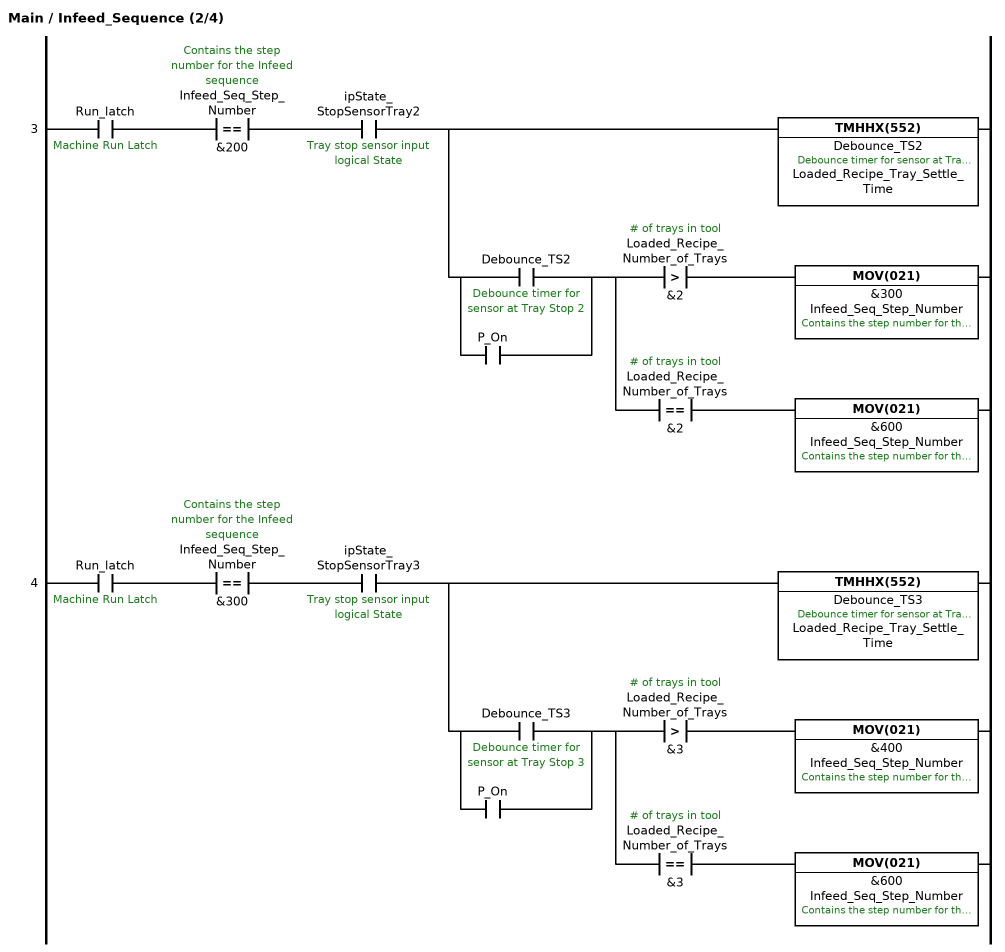
; [picture p24: Main / Infeed_Sequence, rungs 3-4]
; rung 3
LD Run_latch  ; Machine Run Latch
AND=(300) Infeed_Seq_Step_Number &200  ; Contains the step number for the Infeed sequence
AND ipState_StopSensorTray2  ; Tray stop sensor input logical State
TMHHX(552) Debounce_TS2 Loaded_Recipe_Tray_Settle_Time  ; Debounce timer for sensor at Tray Stop 2
LD Debounce_TS2  ; Debounce timer for sensor at Tray Stop 2
OR P_On  // Sensor on and off filters added elsewhere.  Bypassed on 9/25/14 per Gary Liles.
ANDLD
OUT TR0
AND>(320) Loaded_Recipe_Number_of_Trays &2  ; # of trays in tool
MOV(021) &300 Infeed_Seq_Step_Number  ; Contains the step number for the Infeed sequence
LD TR0
AND=(300) Loaded_Recipe_Number_of_Trays &2  ; # of trays in tool
MOV(021) &600 Infeed_Seq_Step_Number  ; Contains the step number for the Infeed sequence
; rung 4
LD Run_latch  ; Machine Run Latch
AND=(300) Infeed_Seq_Step_Number &300  ; Contains the step number for the Infeed sequence
AND ipState_StopSensorTray3  ; Tray stop sensor input logical State
TMHHX(552) Debounce_TS3 Loaded_Recipe_Tray_Settle_Time  ; Debounce timer for sensor at Tray Stop 3
LD Debounce_TS3  ; Debounce timer for sensor at Tray Stop 3
OR P_On  // Sensor on and off filters added elsewhere.  Bypassed on 9/25/14 per Gary Liles.
ANDLD
OUT TR0
AND>(320) Loaded_Recipe_Number_of_Trays &3  ; # of trays in tool
MOV(021) &400 Infeed_Seq_Step_Number  ; Contains the step number for the Infeed sequence
LD TR0
AND=(300) Loaded_Recipe_Number_of_Trays &3  ; # of trays in tool
MOV(021) &600 Infeed_Seq_Step_Number  ; Contains the step number for the Infeed sequence

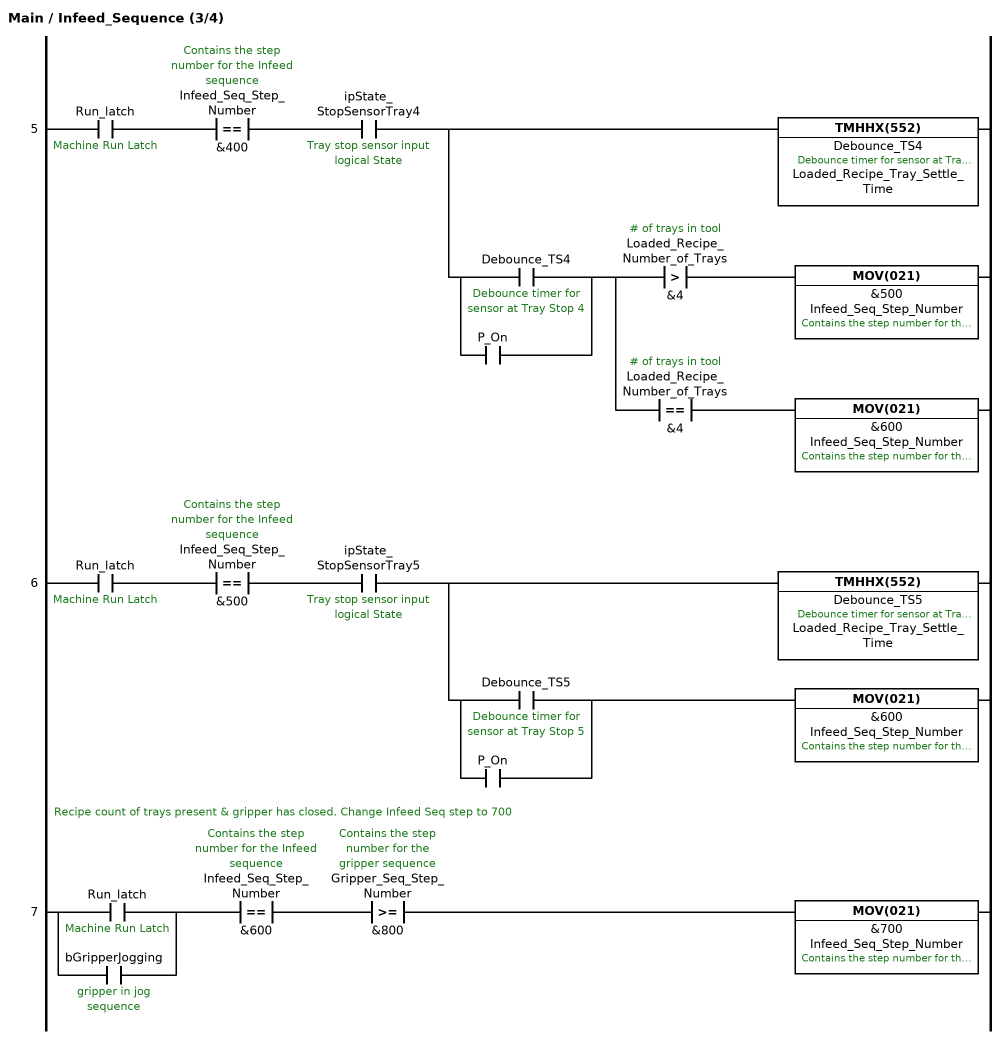
; rung 5
LD Run_latch  ; Machine Run Latch
AND=(300) Infeed_Seq_Step_Number &400  ; Contains the step number for the Infeed sequence
AND ipState_StopSensorTray4  ; Tray stop sensor input logical State
TMHHX(552) Debounce_TS4 Loaded_Recipe_Tray_Settle_Time  ; Debounce timer for sensor at Tray Stop 4
LD Debounce_TS4  ; Debounce timer for sensor at Tray Stop 4
OR P_On  // Sensor on and off filters added elsewhere.  Bypassed on 9/25/14 per Gary Liles.
ANDLD
OUT TR0
AND>(320) Loaded_Recipe_Number_of_Trays &4  ; # of trays in tool
MOV(021) &500 Infeed_Seq_Step_Number  ; Contains the step number for the Infeed sequence
LD TR0
AND=(300) Loaded_Recipe_Number_of_Trays &4  ; # of trays in tool
MOV(021) &600 Infeed_Seq_Step_Number  ; Contains the step number for the Infeed sequence
; rung 6
LD Run_latch  ; Machine Run Latch
AND=(300) Infeed_Seq_Step_Number &500  ; Contains the step number for the Infeed sequence
AND ipState_StopSensorTray5  ; Tray stop sensor input logical State
TMHHX(552) Debounce_TS5 Loaded_Recipe_Tray_Settle_Time  ; Debounce timer for sensor at Tray Stop 5
LD Debounce_TS5  ; Debounce timer for sensor at Tray Stop 5
OR P_On  // Sensor on and off filters added elsewhere.  Bypassed on 9/25/14 per Gary Liles.
ANDLD
MOV(021) &600 Infeed_Seq_Step_Number  ; Contains the step number for the Infeed sequence
; rung 7: Recipe count of trays present & gripper has closed. Change Infeed Seq step to 700
LD Run_latch  ; Machine Run Latch
OR bGripperJogging  ; gripper in jog sequence
AND=(300) Infeed_Seq_Step_Number &600  ; Contains the step number for the Infeed sequence
AND>=(325) Gripper_Seq_Step_Number &800  ; Contains the step number for the gripper sequence
MOV(021) &700 Infeed_Seq_Step_Number  ; Contains the step number for the Infeed sequence

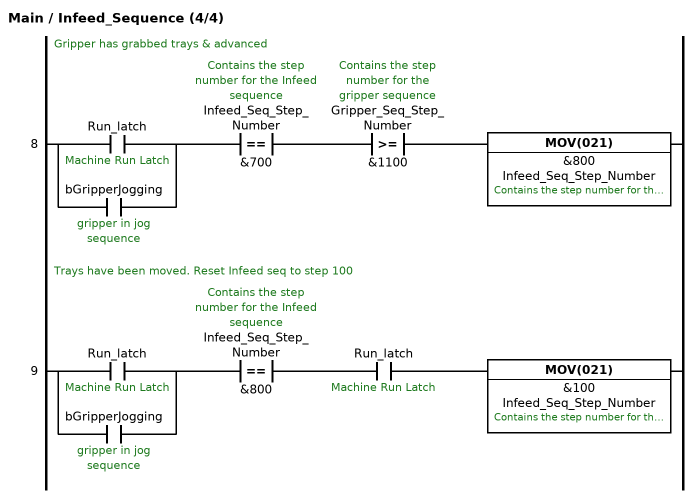
; rung 8: Gripper has grabbed trays & advanced
LD Run_latch  ; Machine Run Latch
OR bGripperJogging  ; gripper in jog sequence
AND=(300) Infeed_Seq_Step_Number &700  ; Contains the step number for the Infeed sequence
AND>=(325) Gripper_Seq_Step_Number &1100  ; Contains the step number for the gripper sequence
MOV(021) &800 Infeed_Seq_Step_Number  ; Contains the step number for the Infeed sequence
; rung 9: Trays have been moved. Reset Infeed seq to step 100
LD Run_latch  ; Machine Run Latch
OR bGripperJogging  ; gripper in jog sequence
AND=(300) Infeed_Seq_Step_Number &800  ; Contains the step number for the Infeed sequence
AND Run_latch  ; Machine Run Latch
MOV(021) &100 Infeed_Seq_Step_Number  ; Contains the step number for the Infeed sequence

### Section Infeed_outputs

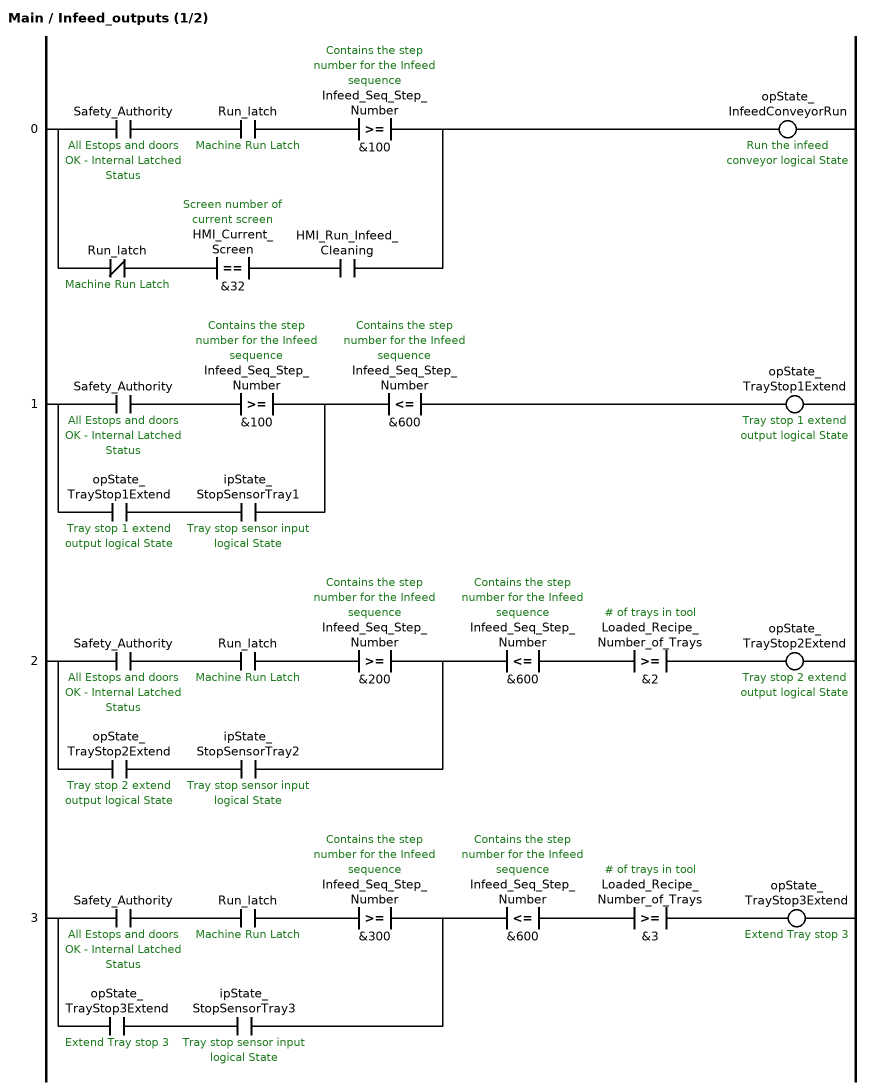
; rung 0
LD Safety_Authority  ; All Estops and doors OK - Internal Latched Status
AND Run_latch  ; Machine Run Latch
AND>=(325) Infeed_Seq_Step_Number &100  ; Contains the step number for the Infeed sequence
LDNOT Run_latch  ; Machine Run Latch
AND=(300) HMI_Current_Screen &32  ; Screen number of current screen
AND HMI_Run_Infeed_Cleaning
ORLD
OUT opState_InfeedConveyorRun  ; Run the infeed conveyor logical State
; rung 1
LD Safety_Authority  ; All Estops and doors OK - Internal Latched Status
AND>=(325) Infeed_Seq_Step_Number &100  ; Contains the step number for the Infeed sequence
LD opState_TrayStop1Extend  ; Tray stop 1 extend output logical State
AND ipState_StopSensorTray1  ; Tray stop sensor input logical State
ORLD
AND<=(315) Infeed_Seq_Step_Number &600  ; Contains the step number for the Infeed sequence
OUT opState_TrayStop1Extend  ; Tray stop 1 extend output logical State
; rung 2
LD Safety_Authority  ; All Estops and doors OK - Internal Latched Status
AND Run_latch  ; Machine Run Latch
AND>=(325) Infeed_Seq_Step_Number &200  ; Contains the step number for the Infeed sequence
LD opState_TrayStop2Extend  ; Tray stop 2 extend output logical State
AND ipState_StopSensorTray2  ; Tray stop sensor input logical State
ORLD
AND<=(315) Infeed_Seq_Step_Number &600  ; Contains the step number for the Infeed sequence
AND>=(325) Loaded_Recipe_Number_of_Trays &2  ; # of trays in tool
OUT opState_TrayStop2Extend  ; Tray stop 2 extend output logical State
; rung 3
LD Safety_Authority  ; All Estops and doors OK - Internal Latched Status
AND Run_latch  ; Machine Run Latch
AND>=(325) Infeed_Seq_Step_Number &300  ; Contains the step number for the Infeed sequence
LD opState_TrayStop3Extend  ; Extend Tray stop 3
AND ipState_StopSensorTray3  ; Tray stop sensor input logical State
ORLD
AND<=(315) Infeed_Seq_Step_Number &600  ; Contains the step number for the Infeed sequence
AND>=(325) Loaded_Recipe_Number_of_Trays &3  ; # of trays in tool
OUT opState_TrayStop3Extend  ; Extend Tray stop 3

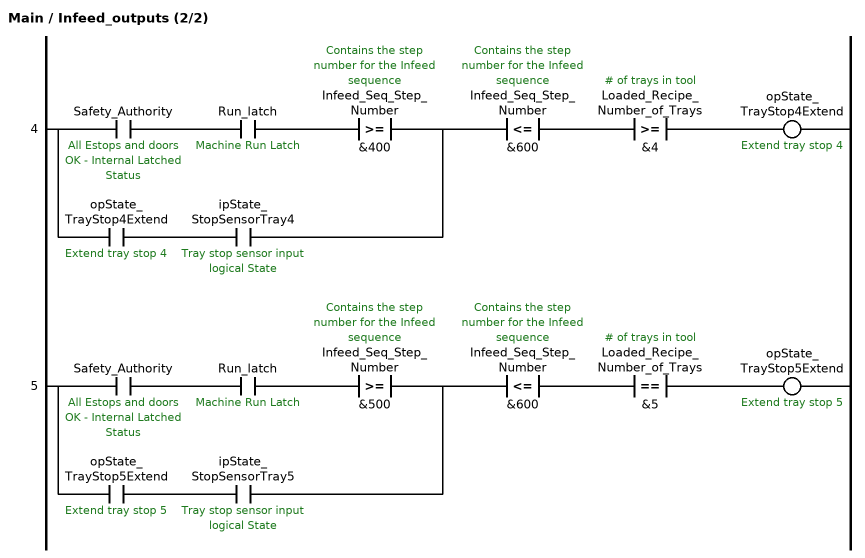
; rung 4
LD Safety_Authority  ; All Estops and doors OK - Internal Latched Status
AND Run_latch  ; Machine Run Latch
AND>=(325) Infeed_Seq_Step_Number &400  ; Contains the step number for the Infeed sequence
LD opState_TrayStop4Extend  ; Extend tray stop 4
AND ipState_StopSensorTray4  ; Tray stop sensor input logical State
ORLD
AND<=(315) Infeed_Seq_Step_Number &600  ; Contains the step number for the Infeed sequence
AND>=(325) Loaded_Recipe_Number_of_Trays &4  ; # of trays in tool
OUT opState_TrayStop4Extend  ; Extend tray stop 4
; rung 5
LD Safety_Authority  ; All Estops and doors OK - Internal Latched Status
AND Run_latch  ; Machine Run Latch
AND>=(325) Infeed_Seq_Step_Number &500  ; Contains the step number for the Infeed sequence
LD opState_TrayStop5Extend  ; Extend tray stop 5
AND ipState_StopSensorTray5  ; Tray stop sensor input logical State
ORLD
AND<=(315) Infeed_Seq_Step_Number &600  ; Contains the step number for the Infeed sequence
AND=(300) Loaded_Recipe_Number_of_Trays &5  ; # of trays in tool
OUT opState_TrayStop5Extend  ; Extend tray stop 5

### Section Grip_Sequence

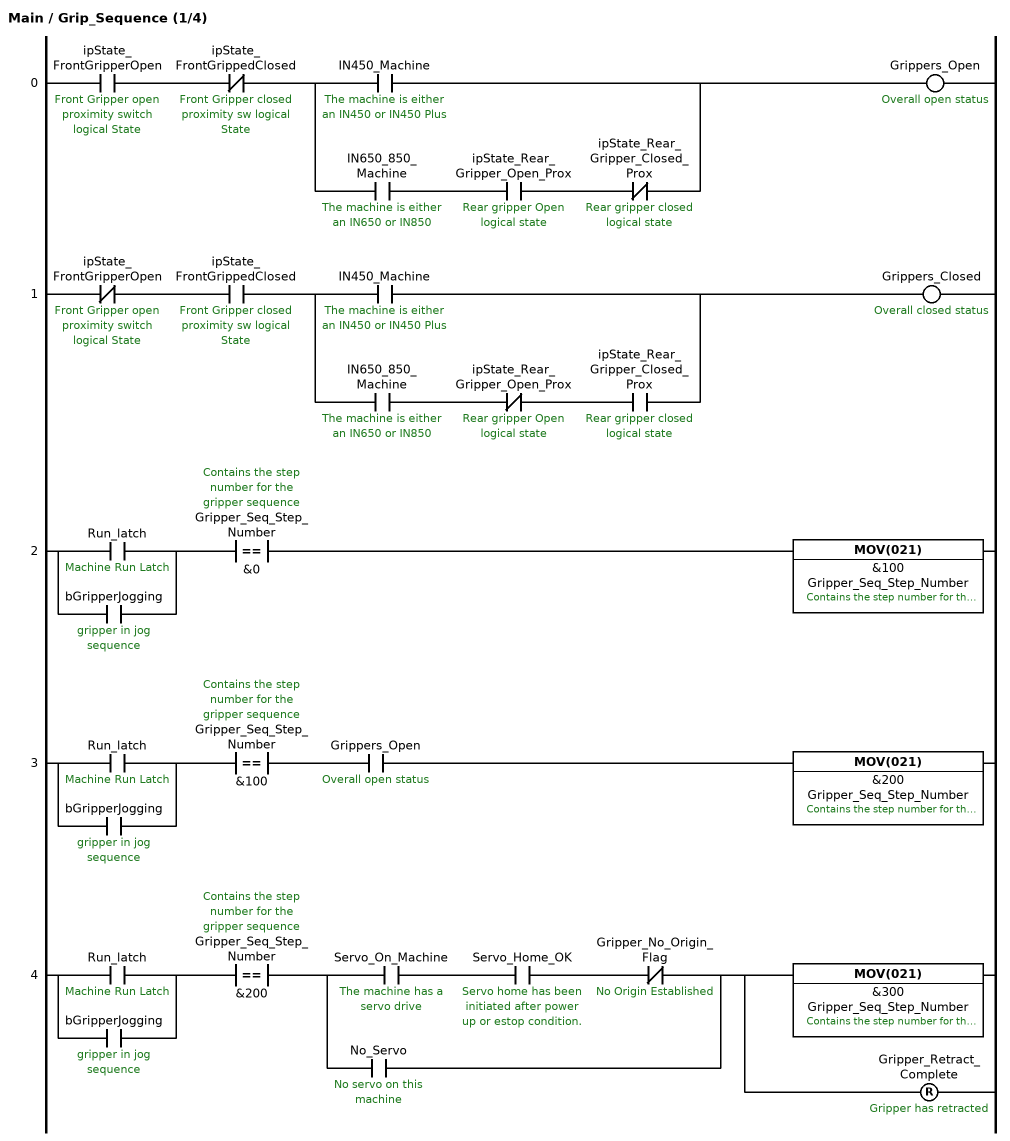
; rung 0
LD ipState_FrontGripperOpen  ; Front Gripper open proximity switch logical State
ANDNOT ipState_FrontGrippedClosed  ; Front Gripper closed proximity sw logical State
LD IN450_Machine  ; The machine is either an IN450 or IN450 Plus
LD IN650_850_Machine  ; The machine is either an IN650 or IN850
AND ipState_Rear_Gripper_Open_Prox  ; Rear gripper Open logical state
ANDNOT ipState_Rear_Gripper_Closed_Prox  ; Rear gripper closed logical state
ORLD
ANDLD
OUT Grippers_Open  ; Overall open status
; rung 1
LDNOT ipState_FrontGripperOpen  ; Front Gripper open proximity switch logical State
AND ipState_FrontGrippedClosed  ; Front Gripper closed proximity sw logical State
LD IN450_Machine  ; The machine is either an IN450 or IN450 Plus
LD IN650_850_Machine  ; The machine is either an IN650 or IN850
ANDNOT ipState_Rear_Gripper_Open_Prox  ; Rear gripper Open logical state
AND ipState_Rear_Gripper_Closed_Prox  ; Rear gripper closed logical state
ORLD
ANDLD
OUT Grippers_Closed  ; Overall closed status
; rung 2
LD Run_latch  ; Machine Run Latch
OR bGripperJogging  ; gripper in jog sequence
AND=(300) Gripper_Seq_Step_Number &0  ; Contains the step number for the gripper sequence
MOV(021) &100 Gripper_Seq_Step_Number  ; Contains the step number for the gripper sequence
; rung 3
LD Run_latch  ; Machine Run Latch
OR bGripperJogging  ; gripper in jog sequence
AND=(300) Gripper_Seq_Step_Number &100  ; Contains the step number for the gripper sequence
AND Grippers_Open  ; Overall open status
MOV(021) &200 Gripper_Seq_Step_Number  ; Contains the step number for the gripper sequence
; rung 4
LD Run_latch  ; Machine Run Latch
OR bGripperJogging  ; gripper in jog sequence
AND=(300) Gripper_Seq_Step_Number &200  ; Contains the step number for the gripper sequence
LD Servo_On_Machine  ; The machine has a servo drive
AND Servo_Home_OK  ; Servo home has been initiated after power up or estop condition.
ANDNOT Gripper_No_Origin_Flag  ; No Origin Established
OR No_Servo  ; No servo on this machine
ANDLD
MOV(021) &300 Gripper_Seq_Step_Number  ; Contains the step number for the gripper sequence
RSET Gripper_Retract_Complete  ; Gripper has retracted

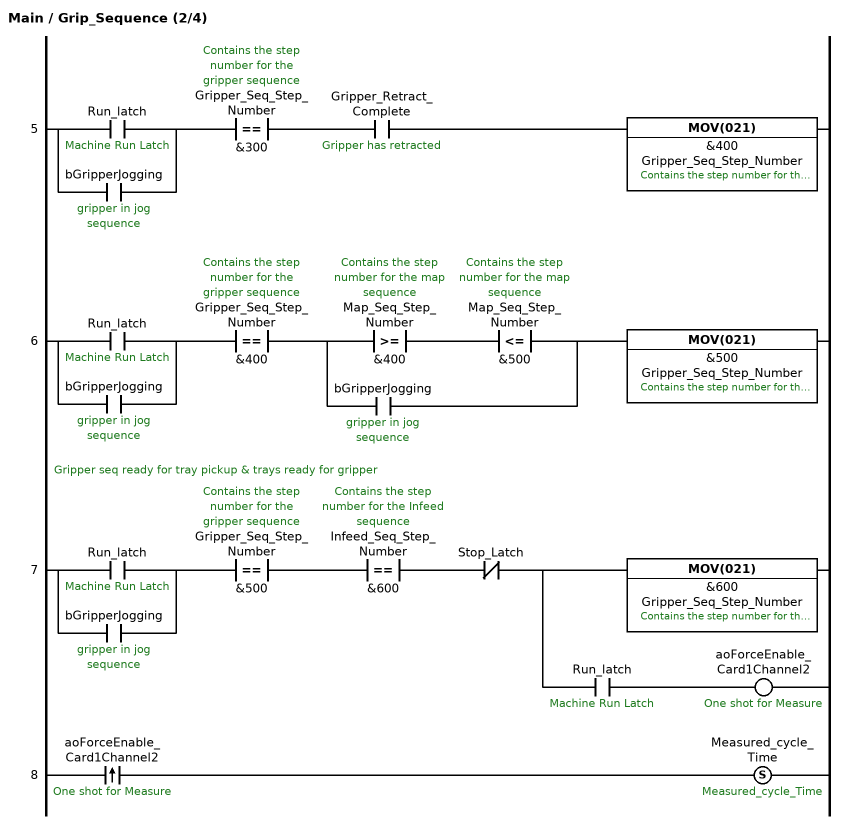
; rung 5
LD Run_latch  ; Machine Run Latch
OR bGripperJogging  ; gripper in jog sequence
AND=(300) Gripper_Seq_Step_Number &300  ; Contains the step number for the gripper sequence
AND Gripper_Retract_Complete  ; Gripper has retracted
MOV(021) &400 Gripper_Seq_Step_Number  ; Contains the step number for the gripper sequence
; rung 6
LD Run_latch  ; Machine Run Latch
OR bGripperJogging  ; gripper in jog sequence
AND=(300) Gripper_Seq_Step_Number &400  ; Contains the step number for the gripper sequence
LD>=(325) Map_Seq_Step_Number &400  ; Contains the step number for the map sequence
AND<=(315) Map_Seq_Step_Number &500  ; Contains the step number for the map sequence
OR bGripperJogging  ; gripper in jog sequence
ANDLD
MOV(021) &500 Gripper_Seq_Step_Number  ; Contains the step number for the gripper sequence
; rung 7: Gripper seq ready for tray pickup & trays ready for gripper
LD Run_latch  ; Machine Run Latch
OR bGripperJogging  ; gripper in jog sequence
AND=(300) Gripper_Seq_Step_Number &500  ; Contains the step number for the gripper sequence
AND=(300) Infeed_Seq_Step_Number &600  ; Contains the step number for the Infeed sequence
ANDNOT Stop_Latch
MOV(021) &600 Gripper_Seq_Step_Number  ; Contains the step number for the gripper sequence
AND Run_latch  ; Machine Run Latch
OUT aoForceEnable_Card1Channel2  ; One shot for Measure
; rung 8
@LD aoForceEnable_Card1Channel2  ; One shot for Measure
SET Measured_cycle_Time  ; Measured_cycle_Time

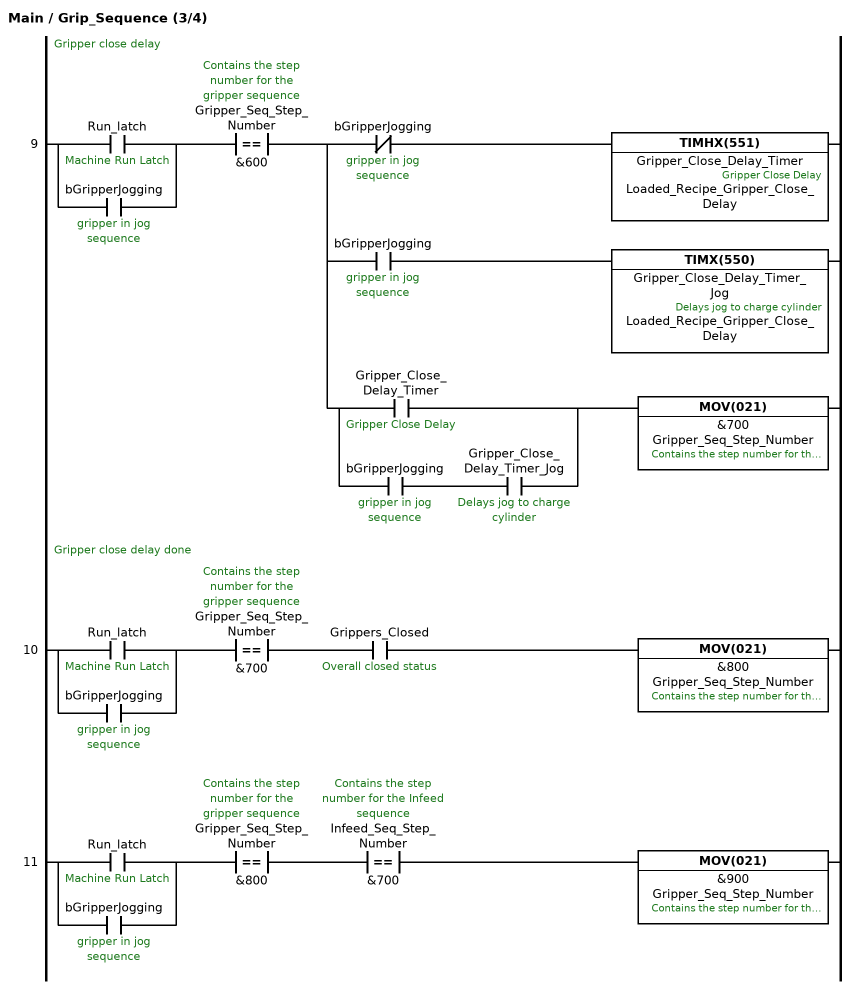
; rung 9: Gripper close delay
LD Run_latch  ; Machine Run Latch
OR bGripperJogging  ; gripper in jog sequence
AND=(300) Gripper_Seq_Step_Number &600  ; Contains the step number for the gripper sequence
OUT TR0
ANDNOT bGripperJogging  ; gripper in jog sequence
TIMHX(551) Gripper_Close_Delay_Timer Loaded_Recipe_Gripper_Close_Delay  ; Gripper Close Delay
LD TR0
AND bGripperJogging  ; gripper in jog sequence
TIMX(550) Gripper_Close_Delay_Timer_Jog Loaded_Recipe_Gripper_Close_Delay  ; Delays jog to charge cylinder
LD TR0
LD Gripper_Close_Delay_Timer  ; Gripper Close Delay
LD bGripperJogging  ; gripper in jog sequence
AND Gripper_Close_Delay_Timer_Jog  ; Delays jog to charge cylinder
ORLD
ANDLD
MOV(021) &700 Gripper_Seq_Step_Number  ; Contains the step number for the gripper sequence
; rung 10: Gripper close delay done
LD Run_latch  ; Machine Run Latch
OR bGripperJogging  ; gripper in jog sequence
AND=(300) Gripper_Seq_Step_Number &700  ; Contains the step number for the gripper sequence
AND Grippers_Closed  ; Overall closed status
MOV(021) &800 Gripper_Seq_Step_Number  ; Contains the step number for the gripper sequence
; rung 11
LD Run_latch  ; Machine Run Latch
OR bGripperJogging  ; gripper in jog sequence
AND=(300) Gripper_Seq_Step_Number &800  ; Contains the step number for the gripper sequence
AND=(300) Infeed_Seq_Step_Number &700  ; Contains the step number for the Infeed sequence
MOV(021) &900 Gripper_Seq_Step_Number  ; Contains the step number for the gripper sequence

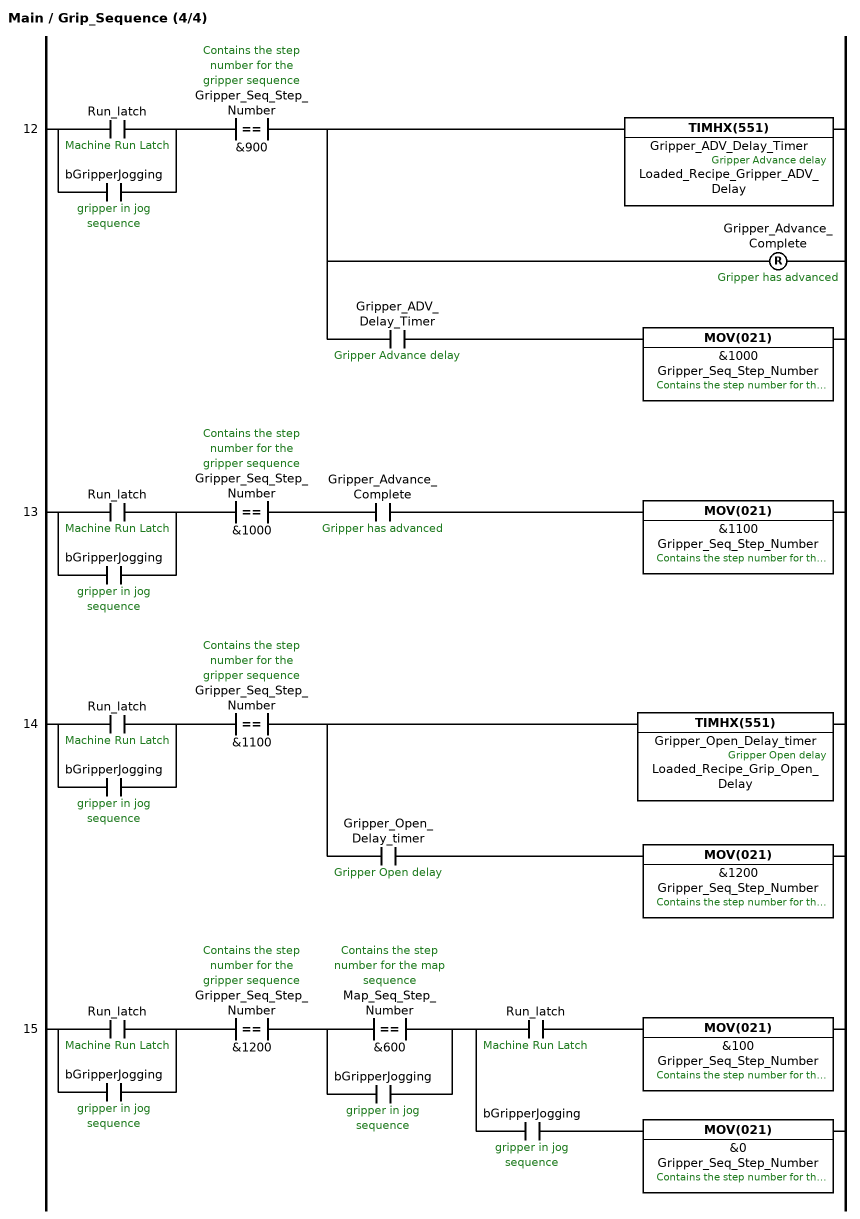
; rung 12
LD Run_latch  ; Machine Run Latch
OR bGripperJogging  ; gripper in jog sequence
AND=(300) Gripper_Seq_Step_Number &900  ; Contains the step number for the gripper sequence
TIMHX(551) Gripper_ADV_Delay_Timer Loaded_Recipe_Gripper_ADV_Delay  ; Gripper Advance delay
RSET Gripper_Advance_Complete  ; Gripper has advanced
AND Gripper_ADV_Delay_Timer  ; Gripper Advance delay
MOV(021) &1000 Gripper_Seq_Step_Number  ; Contains the step number for the gripper sequence
; rung 13
LD Run_latch  ; Machine Run Latch
OR bGripperJogging  ; gripper in jog sequence
AND=(300) Gripper_Seq_Step_Number &1000  ; Contains the step number for the gripper sequence
AND Gripper_Advance_Complete  ; Gripper has advanced
MOV(021) &1100 Gripper_Seq_Step_Number  ; Contains the step number for the gripper sequence
; rung 14
LD Run_latch  ; Machine Run Latch
OR bGripperJogging  ; gripper in jog sequence
AND=(300) Gripper_Seq_Step_Number &1100  ; Contains the step number for the gripper sequence
TIMHX(551) Gripper_Open_Delay_timer Loaded_Recipe_Grip_Open_Delay  ; Gripper Open delay
AND Gripper_Open_Delay_timer  ; Gripper Open delay
MOV(021) &1200 Gripper_Seq_Step_Number  ; Contains the step number for the gripper sequence
; rung 15
LD Run_latch  ; Machine Run Latch
OR bGripperJogging  ; gripper in jog sequence
AND=(300) Gripper_Seq_Step_Number &1200  ; Contains the step number for the gripper sequence
LD=(300) Map_Seq_Step_Number &600  ; Contains the step number for the map sequence
OR bGripperJogging  ; gripper in jog sequence
ANDLD
OUT TR0
AND Run_latch  ; Machine Run Latch
MOV(021) &100 Gripper_Seq_Step_Number  ; Contains the step number for the gripper sequence
LD TR0
AND bGripperJogging  ; gripper in jog sequence
MOV(021) &0 Gripper_Seq_Step_Number  ; Contains the step number for the gripper sequence

### Section Grip_Outputs

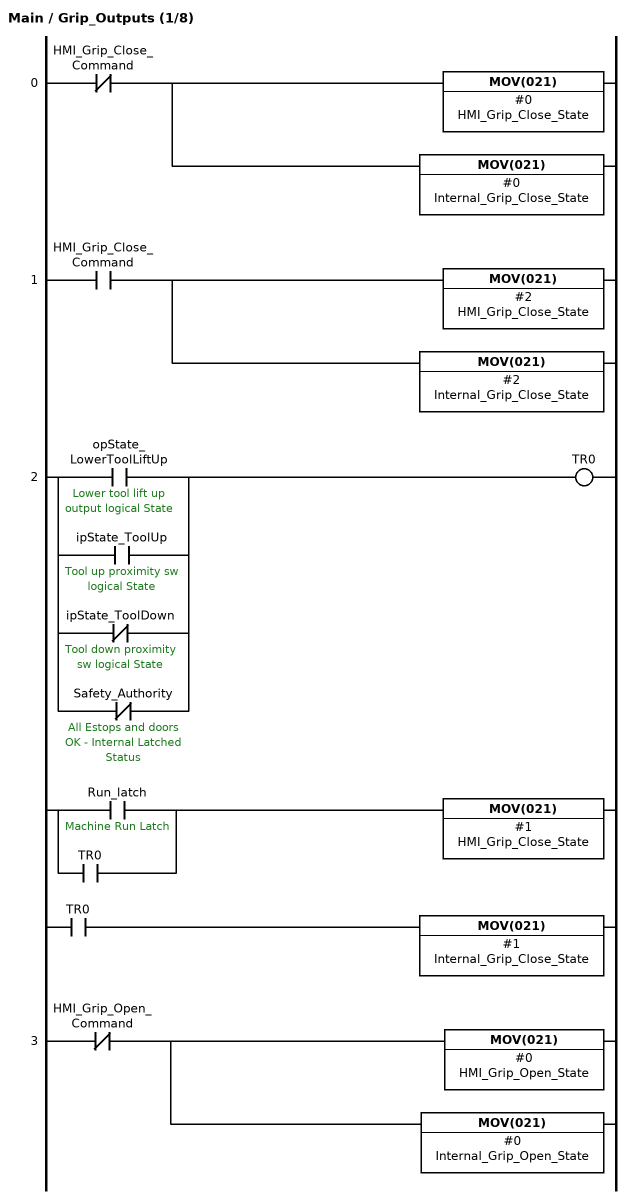
; rung 0
LDNOT HMI_Grip_Close_Command
MOV(021) #0 HMI_Grip_Close_State
MOV(021) #0 Internal_Grip_Close_State
; rung 1
LD HMI_Grip_Close_Command
MOV(021) #2 HMI_Grip_Close_State
MOV(021) #2 Internal_Grip_Close_State
; rung 2
LD Run_latch  ; Machine Run Latch
LD opState_LowerToolLiftUp  ; Lower tool lift up output logical State
OR ipState_ToolUp  ; Tool up proximity sw logical State
ORNOT ipState_ToolDown  ; Tool down proximity sw logical State
ORNOT Safety_Authority  ; All Estops and doors OK - Internal Latched Status
OUT TR0
ORLD
MOV(021) #1 HMI_Grip_Close_State
LD TR0
MOV(021) #1 Internal_Grip_Close_State
; rung 3
LDNOT HMI_Grip_Open_Command
MOV(021) #0 HMI_Grip_Open_State
MOV(021) #0 Internal_Grip_Open_State

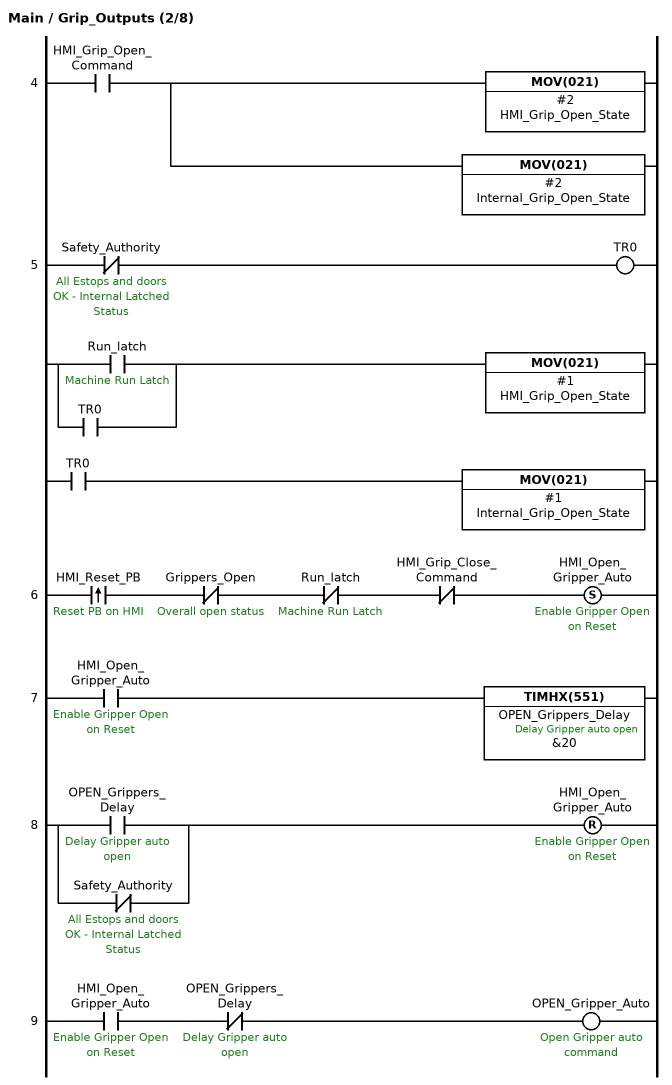
; rung 4
LD HMI_Grip_Open_Command
MOV(021) #2 HMI_Grip_Open_State
MOV(021) #2 Internal_Grip_Open_State
; rung 5
LD Run_latch  ; Machine Run Latch
LDNOT Safety_Authority  ; All Estops and doors OK - Internal Latched Status
OUT TR0
ORLD
MOV(021) #1 HMI_Grip_Open_State
LD TR0
MOV(021) #1 Internal_Grip_Open_State
; rung 6
@LD HMI_Reset_PB  ; Reset PB on HMI
ANDNOT Grippers_Open  ; Overall open status
ANDNOT Run_latch  ; Machine Run Latch
ANDNOT HMI_Grip_Close_Command
SET HMI_Open_Gripper_Auto  ; Enable Gripper Open on Reset
; rung 7
LD HMI_Open_Gripper_Auto  ; Enable Gripper Open on Reset
TIMHX(551) OPEN_Grippers_Delay &20  ; Delay Gripper auto open
; rung 8
LD OPEN_Grippers_Delay  ; Delay Gripper auto open
ORNOT Safety_Authority  ; All Estops and doors OK - Internal Latched Status
RSET HMI_Open_Gripper_Auto  ; Enable Gripper Open on Reset
; rung 9
LD HMI_Open_Gripper_Auto  ; Enable Gripper Open on Reset
ANDNOT OPEN_Grippers_Delay  ; Delay Gripper auto open
OUT OPEN_Gripper_Auto  ; Open Gripper auto command

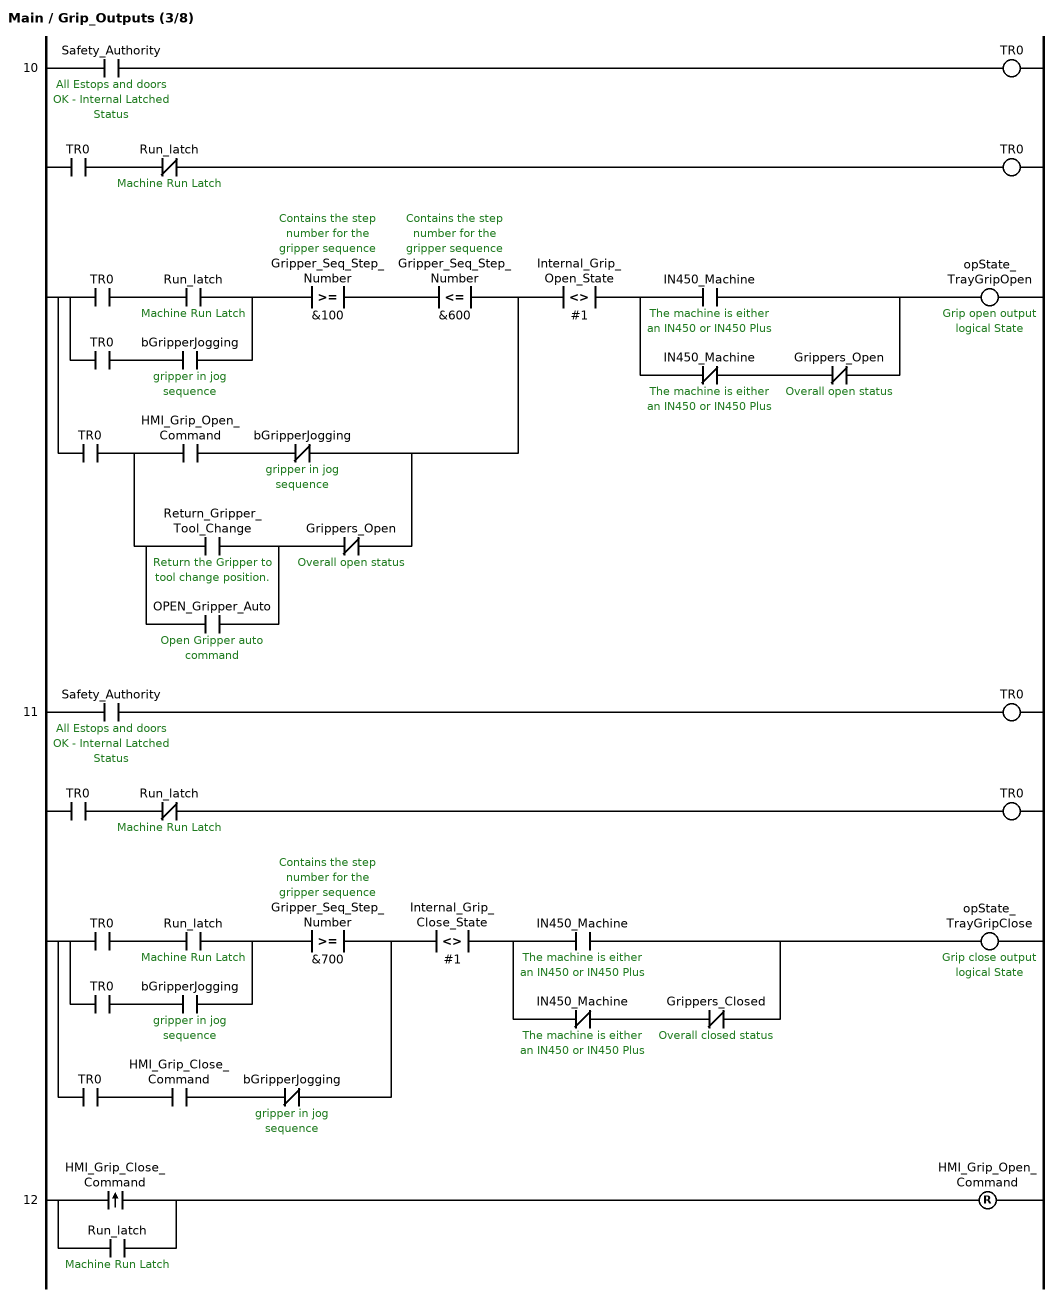
; rung 10
LD Safety_Authority  ; All Estops and doors OK - Internal Latched Status
OUT TR0
AND Run_latch  ; Machine Run Latch
LD TR0
ANDNOT Run_latch  ; Machine Run Latch
OUT TR0
AND bGripperJogging  ; gripper in jog sequence
ORLD
AND>=(325) Gripper_Seq_Step_Number &100  ; Contains the step number for the gripper sequence
AND<=(315) Gripper_Seq_Step_Number &600  ; Contains the step number for the gripper sequence
LD TR0
LD HMI_Grip_Open_Command
ANDNOT bGripperJogging  ; gripper in jog sequence
LD Return_Gripper_Tool_Change  ; Return the Gripper to tool change position.
OR OPEN_Gripper_Auto  ; Open Gripper auto command
ANDNOT Grippers_Open  ; Overall open status
ORLD
ANDLD
ORLD
AND<>(305) Internal_Grip_Open_State #1
LD IN450_Machine  ; The machine is either an IN450 or IN450 Plus
LDNOT IN450_Machine  ; The machine is either an IN450 or IN450 Plus
ANDNOT Grippers_Open  ; Overall open status
ORLD
ANDLD
OUT opState_TrayGripOpen  ; Grip open output logical State
; rung 11
LD Safety_Authority  ; All Estops and doors OK - Internal Latched Status
OUT TR0
AND Run_latch  ; Machine Run Latch
LD TR0
ANDNOT Run_latch  ; Machine Run Latch
OUT TR0
AND bGripperJogging  ; gripper in jog sequence
ORLD
AND>=(325) Gripper_Seq_Step_Number &700  ; Contains the step number for the gripper sequence
LD TR0
AND HMI_Grip_Close_Command
ANDNOT bGripperJogging  ; gripper in jog sequence
ORLD
AND<>(305) Internal_Grip_Close_State #1
LD IN450_Machine  ; The machine is either an IN450 or IN450 Plus
LDNOT IN450_Machine  ; The machine is either an IN450 or IN450 Plus
ANDNOT Grippers_Closed  ; Overall closed status
ORLD
ANDLD
OUT opState_TrayGripClose  ; Grip close output logical State
; rung 12
@LD HMI_Grip_Close_Command
OR Run_latch  ; Machine Run Latch
RSET HMI_Grip_Open_Command

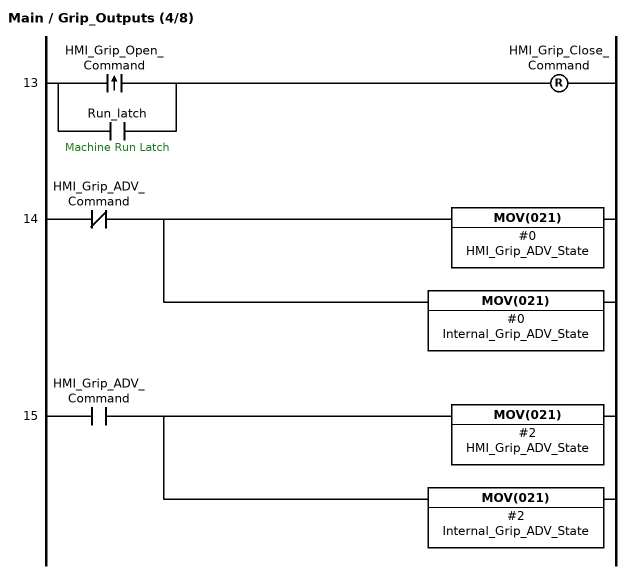
; rung 13
@LD HMI_Grip_Open_Command
OR Run_latch  ; Machine Run Latch
RSET HMI_Grip_Close_Command
; rung 14
LDNOT HMI_Grip_ADV_Command
MOV(021) #0 HMI_Grip_ADV_State
MOV(021) #0 Internal_Grip_ADV_State
; rung 15
LD HMI_Grip_ADV_Command
MOV(021) #2 HMI_Grip_ADV_State
MOV(021) #2 Internal_Grip_ADV_State

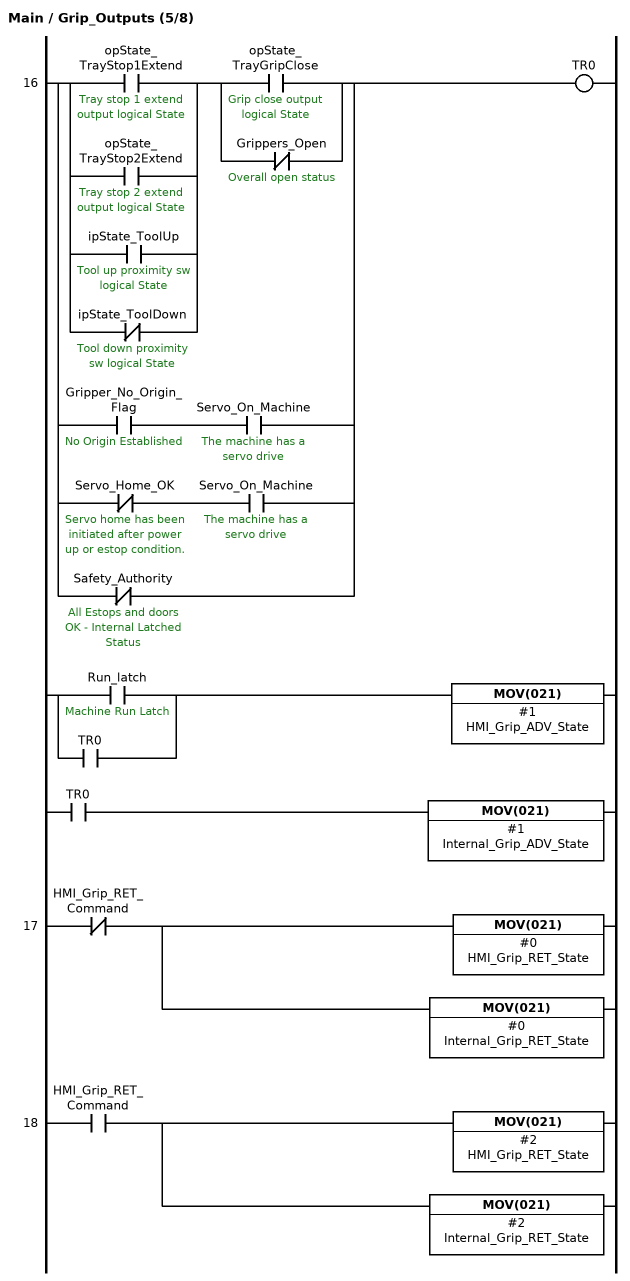
; rung 16
LD Run_latch  ; Machine Run Latch
LD opState_TrayStop1Extend  ; Tray stop 1 extend output logical State
OR opState_TrayStop2Extend  ; Tray stop 2 extend output logical State
OR ipState_ToolUp  ; Tool up proximity sw logical State
ORNOT ipState_ToolDown  ; Tool down proximity sw logical State
LD opState_TrayGripClose  ; Grip close output logical State
ORNOT Grippers_Open  ; Overall open status
ANDLD
LD Gripper_No_Origin_Flag  ; No Origin Established
AND Servo_On_Machine  ; The machine has a servo drive
ORLD
LDNOT Servo_Home_OK  ; Servo home has been initiated after power up or estop condition.
AND Servo_On_Machine  ; The machine has a servo drive
ORLD
ORNOT Safety_Authority  ; All Estops and doors OK - Internal Latched Status
OUT TR0
ORLD
MOV(021) #1 HMI_Grip_ADV_State
LD TR0
MOV(021) #1 Internal_Grip_ADV_State
; rung 17
LDNOT HMI_Grip_RET_Command
MOV(021) #0 HMI_Grip_RET_State
MOV(021) #0 Internal_Grip_RET_State
; rung 18
LD HMI_Grip_RET_Command
MOV(021) #2 HMI_Grip_RET_State
MOV(021) #2 Internal_Grip_RET_State

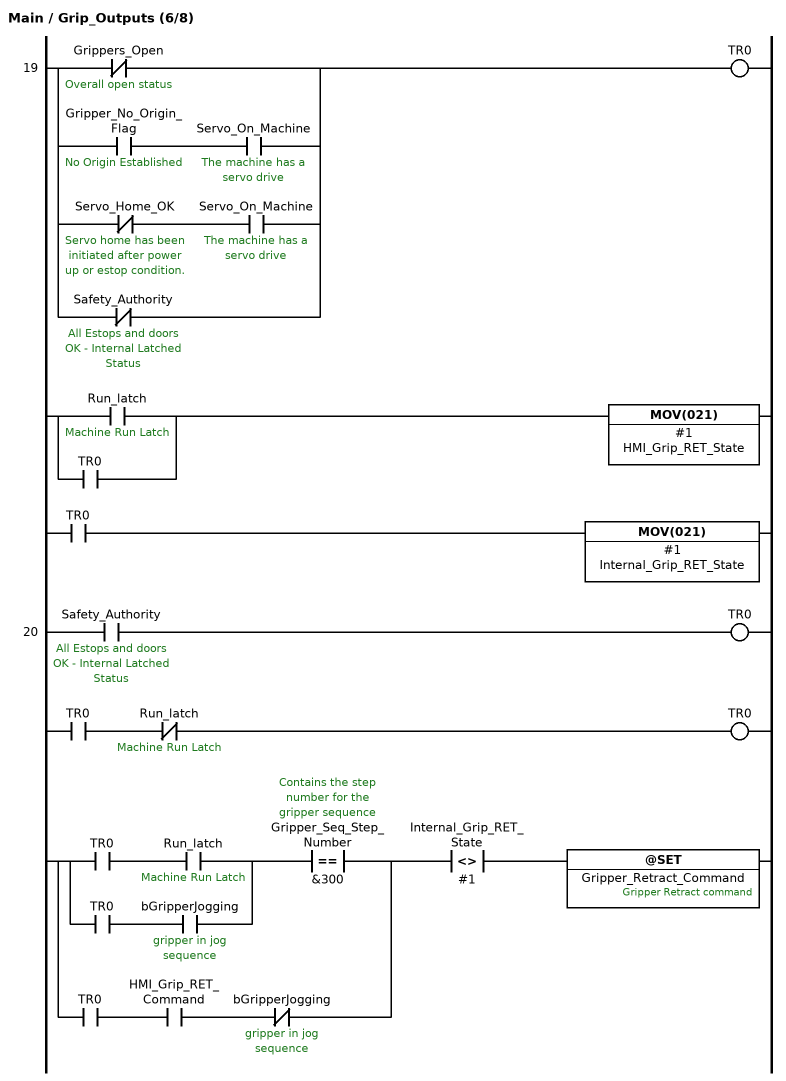
; rung 19
LD Run_latch  ; Machine Run Latch
LDNOT Grippers_Open  ; Overall open status
LD Gripper_No_Origin_Flag  ; No Origin Established
AND Servo_On_Machine  ; The machine has a servo drive
ORLD
LDNOT Servo_Home_OK  ; Servo home has been initiated after power up or estop condition.
AND Servo_On_Machine  ; The machine has a servo drive
ORLD
ORNOT Safety_Authority  ; All Estops and doors OK - Internal Latched Status
OUT TR0
ORLD
MOV(021) #1 HMI_Grip_RET_State
LD TR0
MOV(021) #1 Internal_Grip_RET_State
; rung 20
LD Safety_Authority  ; All Estops and doors OK - Internal Latched Status
OUT TR0
AND Run_latch  ; Machine Run Latch
LD TR0
ANDNOT Run_latch  ; Machine Run Latch
OUT TR0
AND bGripperJogging  ; gripper in jog sequence
ORLD
AND=(300) Gripper_Seq_Step_Number &300  ; Contains the step number for the gripper sequence
LD TR0
AND HMI_Grip_RET_Command
ANDNOT bGripperJogging  ; gripper in jog sequence
ORLD
AND<>(305) Internal_Grip_RET_State #1
@SET Gripper_Retract_Command  ; Gripper Retract command

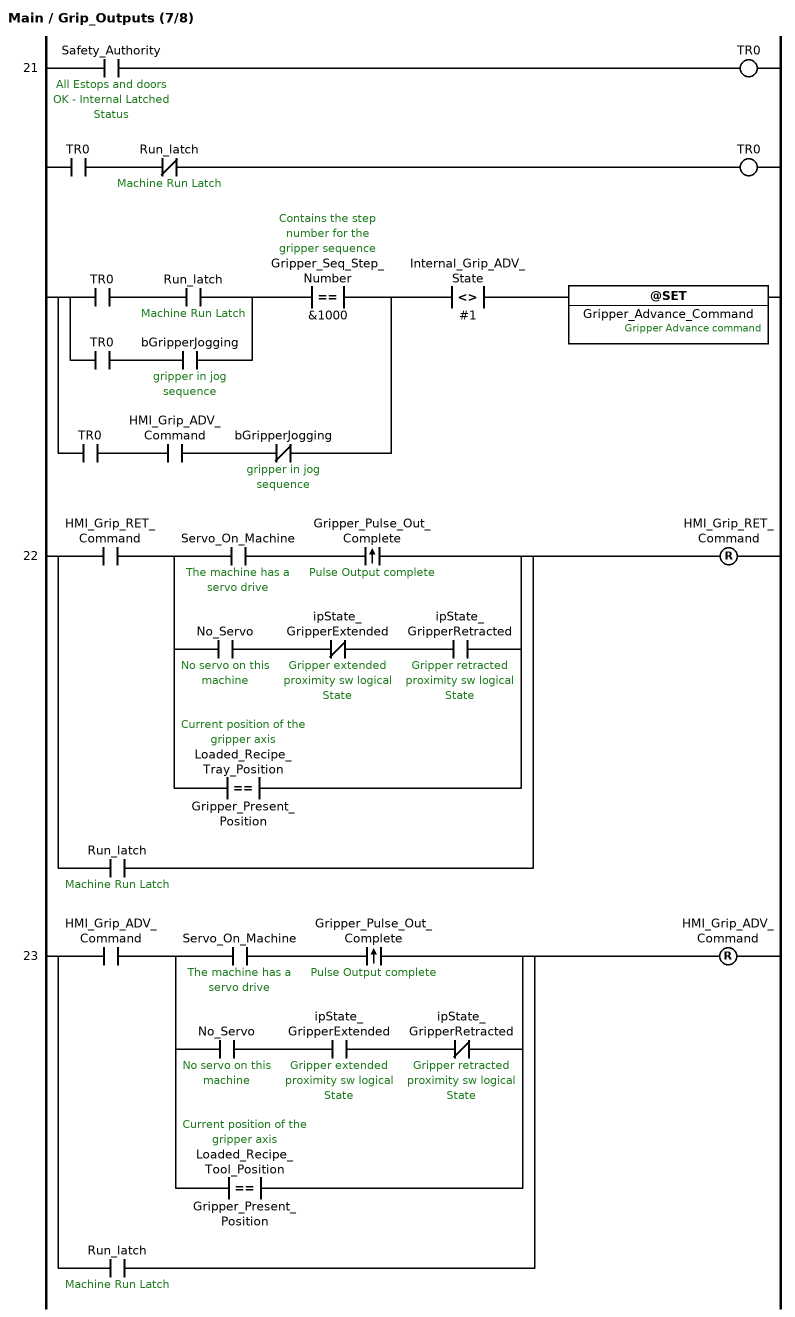
; rung 21
LD Safety_Authority  ; All Estops and doors OK - Internal Latched Status
OUT TR0
AND Run_latch  ; Machine Run Latch
LD TR0
ANDNOT Run_latch  ; Machine Run Latch
OUT TR0
AND bGripperJogging  ; gripper in jog sequence
ORLD
AND=(300) Gripper_Seq_Step_Number &1000  ; Contains the step number for the gripper sequence
LD TR0
AND HMI_Grip_ADV_Command
ANDNOT bGripperJogging  ; gripper in jog sequence
ORLD
AND<>(305) Internal_Grip_ADV_State #1
@SET Gripper_Advance_Command  ; Gripper Advance command
; rung 22
LD HMI_Grip_RET_Command
LD Servo_On_Machine  ; The machine has a servo drive
@AND Gripper_Pulse_Out_Complete  ; Pulse Output complete
LD No_Servo  ; No servo on this machine
ANDNOT ipState_GripperExtended  ; Gripper extended proximity sw logical State
AND ipState_GripperRetracted  ; Gripper retracted proximity sw logical State
ORLD
OR=(300) Loaded_Recipe_Tray_Position Gripper_Present_Position  ; Current position of the gripper axis
ANDLD
OR Run_latch  ; Machine Run Latch
RSET HMI_Grip_RET_Command
; rung 23
LD HMI_Grip_ADV_Command
LD Servo_On_Machine  ; The machine has a servo drive
@AND Gripper_Pulse_Out_Complete  ; Pulse Output complete
LD No_Servo  ; No servo on this machine
AND ipState_GripperExtended  ; Gripper extended proximity sw logical State
ANDNOT ipState_GripperRetracted  ; Gripper retracted proximity sw logical State
ORLD
OR=(300) Loaded_Recipe_Tool_Position Gripper_Present_Position  ; Current position of the gripper axis
ANDLD
OR Run_latch  ; Machine Run Latch
RSET HMI_Grip_ADV_Command

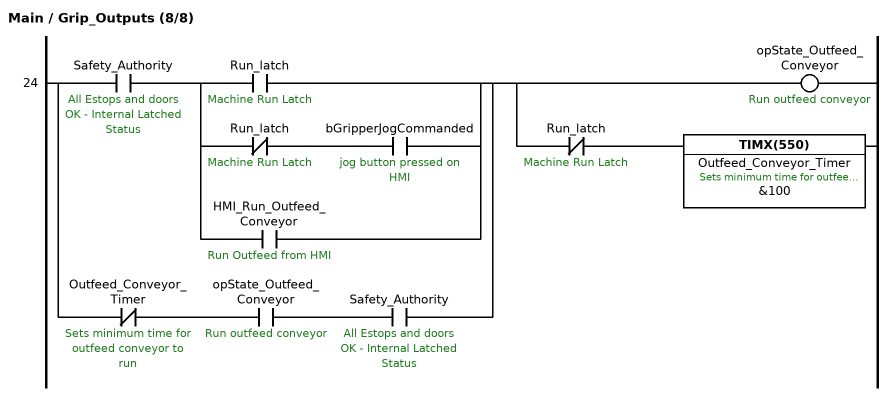
; rung 24
LD Safety_Authority  ; All Estops and doors OK - Internal Latched Status
LD Run_latch  ; Machine Run Latch
LDNOT Run_latch  ; Machine Run Latch
AND bGripperJogCommanded  ; jog button pressed on HMI
ORLD
OR HMI_Run_Outfeed_Conveyor  ; Run Outfeed from HMI
ANDLD
LDNOT Outfeed_Conveyor_Timer  ; Sets minimum time for outfeed conveyor to run
AND opState_Outfeed_Conveyor  ; Run outfeed conveyor
AND Safety_Authority  ; All Estops and doors OK - Internal Latched Status
ORLD
OUT opState_Outfeed_Conveyor  ; Run outfeed conveyor
ANDNOT Run_latch  ; Machine Run Latch
TIMX(550) Outfeed_Conveyor_Timer &100  ; Sets minimum time for outfeed conveyor to run

### Section Infeed_Gate_Sequence

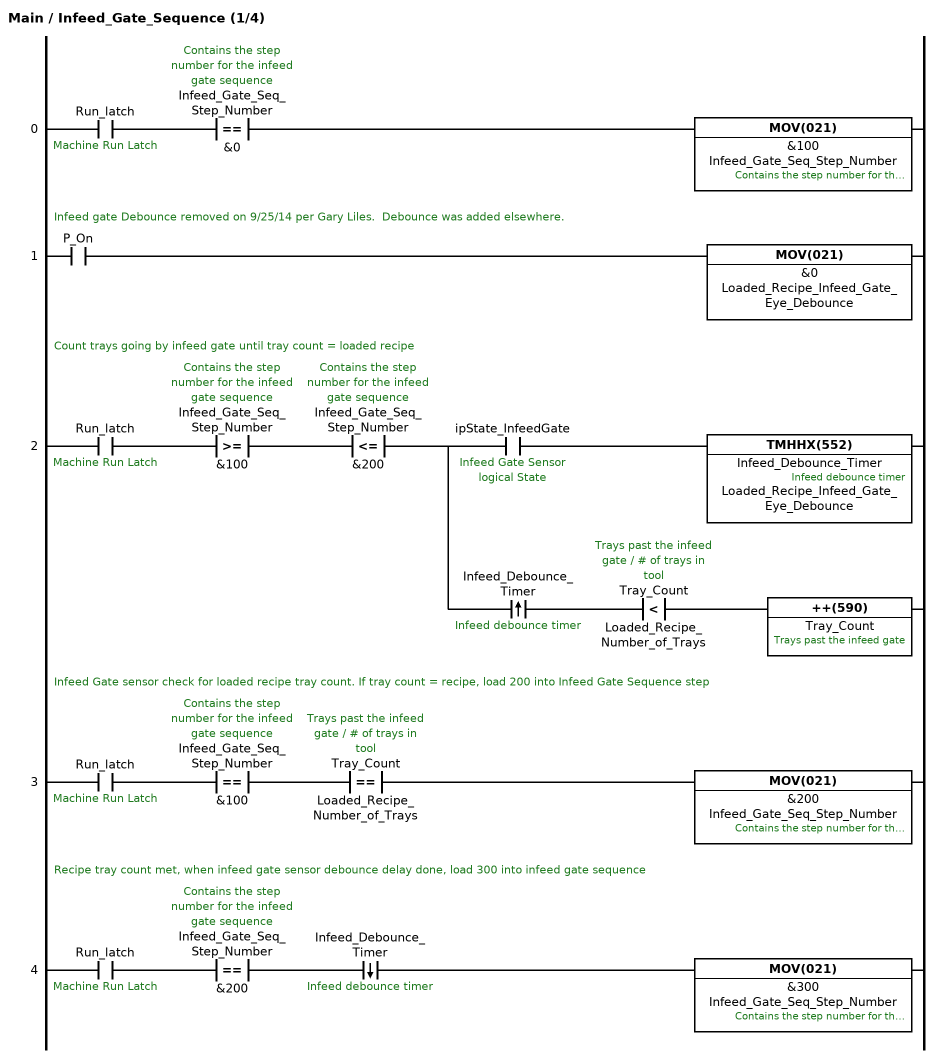
; rung 0
LD Run_latch  ; Machine Run Latch
AND=(300) Infeed_Gate_Seq_Step_Number &0  ; Contains the step number for the infeed gate sequence
MOV(021) &100 Infeed_Gate_Seq_Step_Number  ; Contains the step number for the infeed gate sequence
; rung 1: Infeed gate Debounce removed on 9/25/14 per Gary Liles.  Debounce was added elsewhere.
LD P_On
MOV(021) &0 Loaded_Recipe_Infeed_Gate_Eye_Debounce
; rung 2: Count trays going by infeed gate until tray count = loaded recipe
LD Run_latch  ; Machine Run Latch
AND>=(325) Infeed_Gate_Seq_Step_Number &100  ; Contains the step number for the infeed gate sequence
AND<=(315) Infeed_Gate_Seq_Step_Number &200  ; Contains the step number for the infeed gate sequence
OUT TR0
AND ipState_InfeedGate  ; Infeed Gate Sensor logical State
TMHHX(552) Infeed_Debounce_Timer Loaded_Recipe_Infeed_Gate_Eye_Debounce  ; Infeed debounce timer
LD TR0
@AND Infeed_Debounce_Timer  ; Infeed debounce timer
AND<(310) Tray_Count Loaded_Recipe_Number_of_Trays  ; Trays past the infeed gate, # of trays in tool
++(590) Tray_Count  ; Trays past the infeed gate
; rung 3: Infeed Gate sensor check for loaded recipe tray count. If tray count = recipe, load 200 into Infeed Gate Sequence step
LD Run_latch  ; Machine Run Latch
AND=(300) Infeed_Gate_Seq_Step_Number &100  ; Contains the step number for the infeed gate sequence
AND=(300) Tray_Count Loaded_Recipe_Number_of_Trays  ; Trays past the infeed gate, # of trays in tool
MOV(021) &200 Infeed_Gate_Seq_Step_Number  ; Contains the step number for the infeed gate sequence
; rung 4: Recipe tray count met, when infeed gate sensor debounce delay done, load 300 into infeed gate sequence
LD Run_latch  ; Machine Run Latch
AND=(300) Infeed_Gate_Seq_Step_Number &200  ; Contains the step number for the infeed gate sequence
%AND Infeed_Debounce_Timer  ; Infeed debounce timer
MOV(021) &300 Infeed_Gate_Seq_Step_Number  ; Contains the step number for the infeed gate sequence

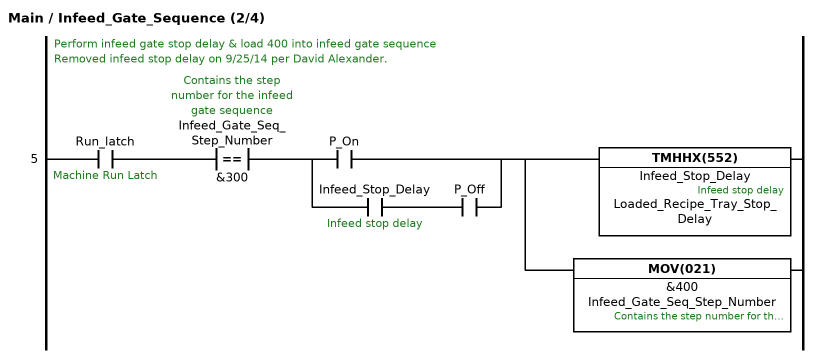
; rung 5: Perform infeed gate stop delay & load 400 into infeed gate sequence / Removed infeed stop delay on 9/25/14 per David Alexander.
LD Run_latch  ; Machine Run Latch
AND=(300) Infeed_Gate_Seq_Step_Number &300  ; Contains the step number for the infeed gate sequence
LD P_On
LD Infeed_Stop_Delay  ; Infeed stop delay
AND P_Off
ORLD
ANDLD
TMHHX(552) Infeed_Stop_Delay Loaded_Recipe_Tray_Stop_Delay  ; Infeed stop delay
MOV(021) &400 Infeed_Gate_Seq_Step_Number  ; Contains the step number for the infeed gate sequence

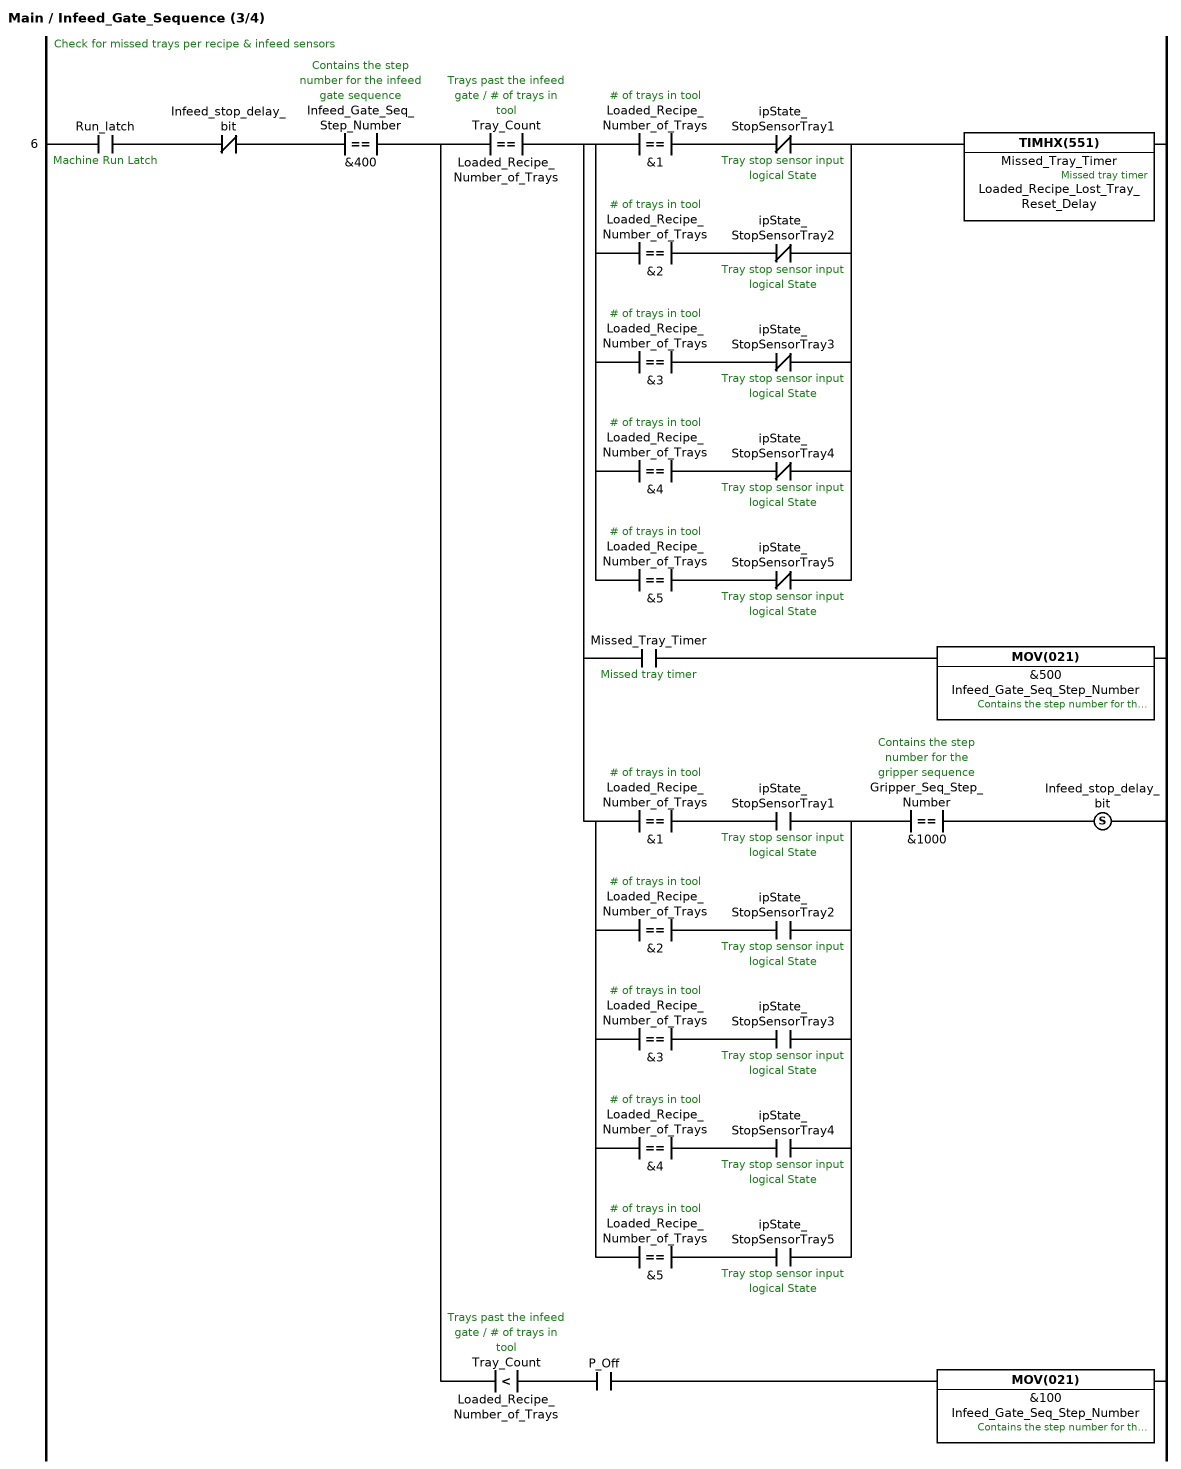
; rung 6: Check for missed trays per recipe & infeed sensors
LD Run_latch  ; Machine Run Latch
ANDNOT Infeed_stop_delay_bit
AND=(300) Infeed_Gate_Seq_Step_Number &400  ; Contains the step number for the infeed gate sequence
OUT TR0
AND=(300) Tray_Count Loaded_Recipe_Number_of_Trays  ; Trays past the infeed gate, # of trays in tool
OUT TR1
LD=(300) Loaded_Recipe_Number_of_Trays &1  ; # of trays in tool
ANDNOT ipState_StopSensorTray1  ; Tray stop sensor input logical State
LD=(300) Loaded_Recipe_Number_of_Trays &2  ; # of trays in tool
ANDNOT ipState_StopSensorTray2  ; Tray stop sensor input logical State
ORLD
LD=(300) Loaded_Recipe_Number_of_Trays &3  ; # of trays in tool
ANDNOT ipState_StopSensorTray3  ; Tray stop sensor input logical State
ORLD
LD=(300) Loaded_Recipe_Number_of_Trays &4  ; # of trays in tool
ANDNOT ipState_StopSensorTray4  ; Tray stop sensor input logical State
ORLD
LD=(300) Loaded_Recipe_Number_of_Trays &5  ; # of trays in tool
ANDNOT ipState_StopSensorTray5  ; Tray stop sensor input logical State
ORLD
ANDLD
TIMHX(551) Missed_Tray_Timer Loaded_Recipe_Lost_Tray_Reset_Delay  ; Missed tray timer
LD TR1
AND Missed_Tray_Timer  ; Missed tray timer
MOV(021) &500 Infeed_Gate_Seq_Step_Number  ; Contains the step number for the infeed gate sequence
LD TR1
LD=(300) Loaded_Recipe_Number_of_Trays &1  ; # of trays in tool
AND ipState_StopSensorTray1  ; Tray stop sensor input logical State
LD=(300) Loaded_Recipe_Number_of_Trays &2  ; # of trays in tool
AND ipState_StopSensorTray2  ; Tray stop sensor input logical State
ORLD
LD=(300) Loaded_Recipe_Number_of_Trays &3  ; # of trays in tool
AND ipState_StopSensorTray3  ; Tray stop sensor input logical State
ORLD
LD=(300) Loaded_Recipe_Number_of_Trays &4  ; # of trays in tool
AND ipState_StopSensorTray4  ; Tray stop sensor input logical State
ORLD
LD=(300) Loaded_Recipe_Number_of_Trays &5  ; # of trays in tool
AND ipState_StopSensorTray5  ; Tray stop sensor input logical State
ORLD
ANDLD
AND=(300) Gripper_Seq_Step_Number &1000  ; Contains the step number for the gripper sequence
SET Infeed_stop_delay_bit
LD TR0
AND<(310) Tray_Count Loaded_Recipe_Number_of_Trays  ; Trays past the infeed gate, # of trays in tool
AND P_Off
MOV(021) &100 Infeed_Gate_Seq_Step_Number  ; Contains the step number for the infeed gate sequence

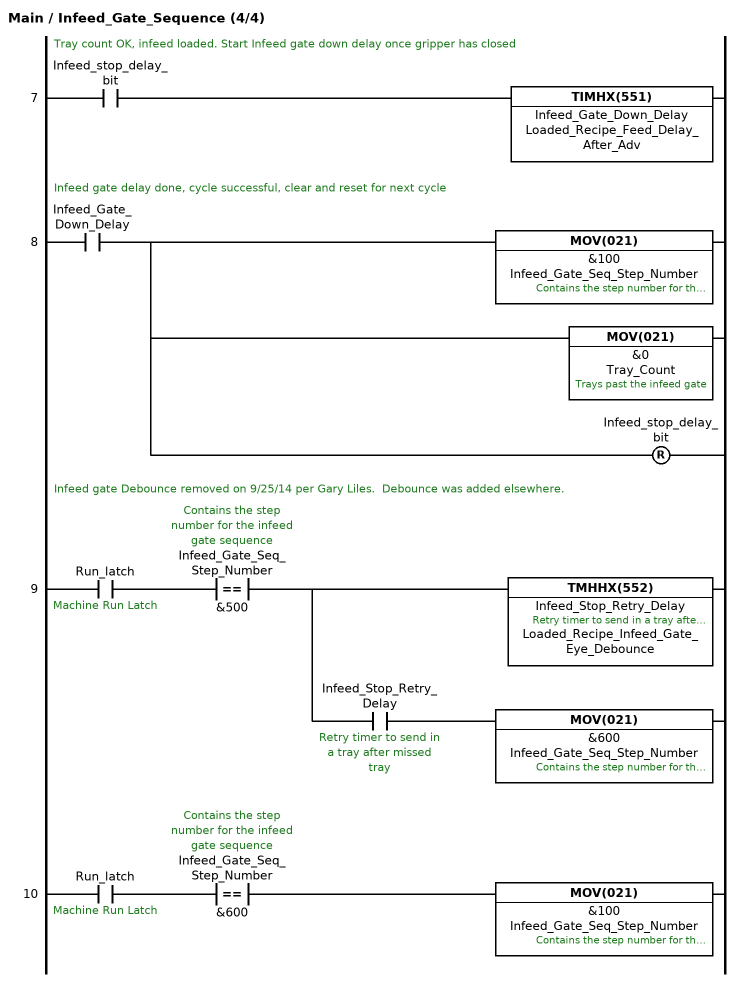
; rung 7: Tray count OK, infeed loaded. Start Infeed gate down delay once gripper has closed
LD Infeed_stop_delay_bit
TIMHX(551) Infeed_Gate_Down_Delay Loaded_Recipe_Feed_Delay_After_Adv
; rung 8: Infeed gate delay done, cycle successful, clear and reset for next cycle
LD Infeed_Gate_Down_Delay
MOV(021) &100 Infeed_Gate_Seq_Step_Number  ; Contains the step number for the infeed gate sequence
MOV(021) &0 Tray_Count  ; Trays past the infeed gate
RSET Infeed_stop_delay_bit
; rung 9: Infeed gate Debounce removed on 9/25/14 per Gary Liles.  Debounce was added elsewhere.
LD Run_latch  ; Machine Run Latch
AND=(300) Infeed_Gate_Seq_Step_Number &500  ; Contains the step number for the infeed gate sequence
TMHHX(552) Infeed_Stop_Retry_Delay Loaded_Recipe_Infeed_Gate_Eye_Debounce  ; Retry timer to send in a tray after missed tray
AND Infeed_Stop_Retry_Delay  ; Retry timer to send in a tray after missed tray
MOV(021) &600 Infeed_Gate_Seq_Step_Number  ; Contains the step number for the infeed gate sequence
; rung 10
LD Run_latch  ; Machine Run Latch
AND=(300) Infeed_Gate_Seq_Step_Number &600  ; Contains the step number for the infeed gate sequence
MOV(021) &100 Infeed_Gate_Seq_Step_Number  ; Contains the step number for the infeed gate sequence

### Section Infeed_Gate_Outputs

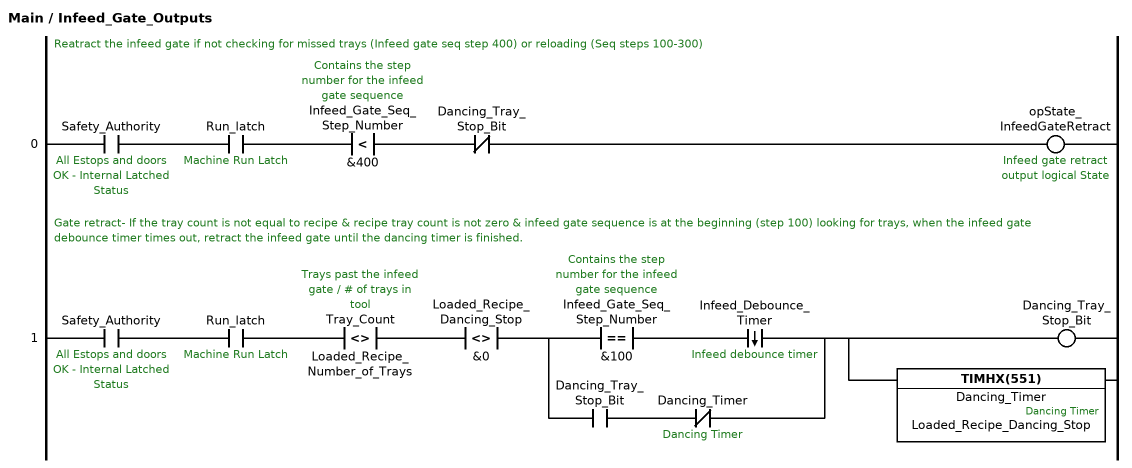
; rung 0: Reatract the infeed gate if not checking for missed trays (Infeed gate seq step 400) or reloading (Seq steps 100-300)
LD Safety_Authority  ; All Estops and doors OK - Internal Latched Status
AND Run_latch  ; Machine Run Latch
AND<(310) Infeed_Gate_Seq_Step_Number &400  ; Contains the step number for the infeed gate sequence
ANDNOT Dancing_Tray_Stop_Bit
OUT opState_InfeedGateRetract  ; Infeed gate retract output logical State
; rung 1: Gate retract- If the tray count is not equal to recipe & recipe tray count is not zero & infeed gate sequence is at the beginning (step 100) looking for trays, when the infeed gate debounce timer times out, retract the infeed gate until the dancing timer is finished.
LD Safety_Authority  ; All Estops and doors OK - Internal Latched Status
AND Run_latch  ; Machine Run Latch
AND<>(305) Tray_Count Loaded_Recipe_Number_of_Trays  ; Trays past the infeed gate, # of trays in tool
AND<>(305) Loaded_Recipe_Dancing_Stop &0
LD=(300) Infeed_Gate_Seq_Step_Number &100  ; Contains the step number for the infeed gate sequence
%AND Infeed_Debounce_Timer  ; Infeed debounce timer
LD Dancing_Tray_Stop_Bit
ANDNOT Dancing_Timer  ; Dancing Timer
ORLD
ANDLD
OUT Dancing_Tray_Stop_Bit
TIMHX(551) Dancing_Timer Loaded_Recipe_Dancing_Stop  ; Dancing Timer

### Section Map_Sequence

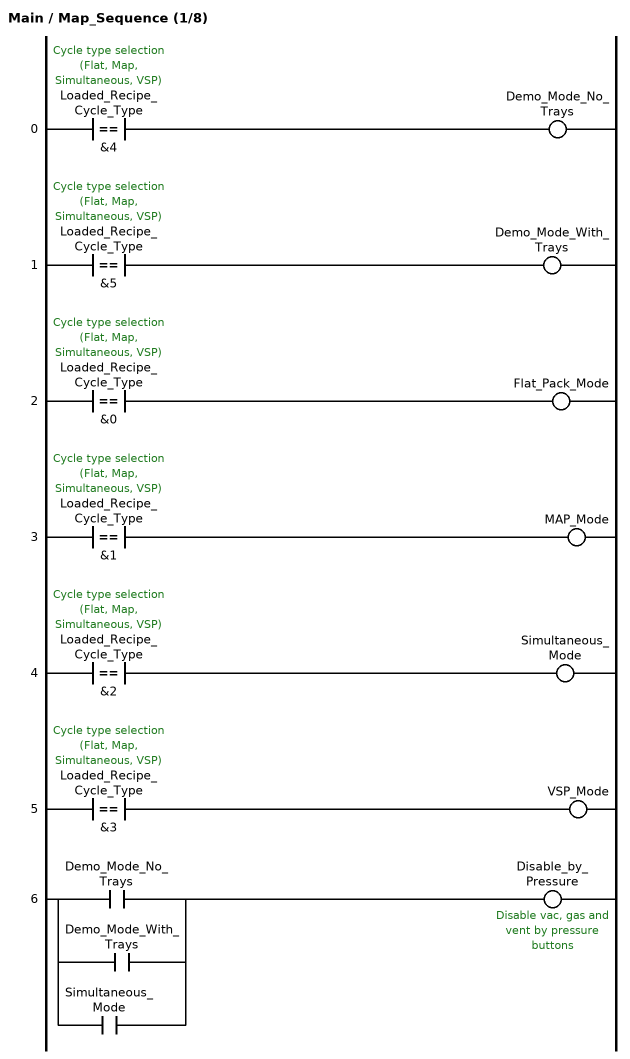
; rung 0
LD=(300) Loaded_Recipe_Cycle_Type &4  ; Cycle type selection (Flat, Map, Simultaneous, VSP)
OUT Demo_Mode_No_Trays
; rung 1
LD=(300) Loaded_Recipe_Cycle_Type &5  ; Cycle type selection (Flat, Map, Simultaneous, VSP)
OUT Demo_Mode_With_Trays
; rung 2
LD=(300) Loaded_Recipe_Cycle_Type &0  ; Cycle type selection (Flat, Map, Simultaneous, VSP)
OUT Flat_Pack_Mode
; rung 3
LD=(300) Loaded_Recipe_Cycle_Type &1  ; Cycle type selection (Flat, Map, Simultaneous, VSP)
OUT MAP_Mode
; rung 4
LD=(300) Loaded_Recipe_Cycle_Type &2  ; Cycle type selection (Flat, Map, Simultaneous, VSP)
OUT Simultaneous_Mode
; rung 5
LD=(300) Loaded_Recipe_Cycle_Type &3  ; Cycle type selection (Flat, Map, Simultaneous, VSP)
OUT VSP_Mode
; rung 6
LD Demo_Mode_No_Trays
OR Demo_Mode_With_Trays
OR Simultaneous_Mode
OUT Disable_by_Pressure  ; Disable vac, gas and vent by pressure buttons

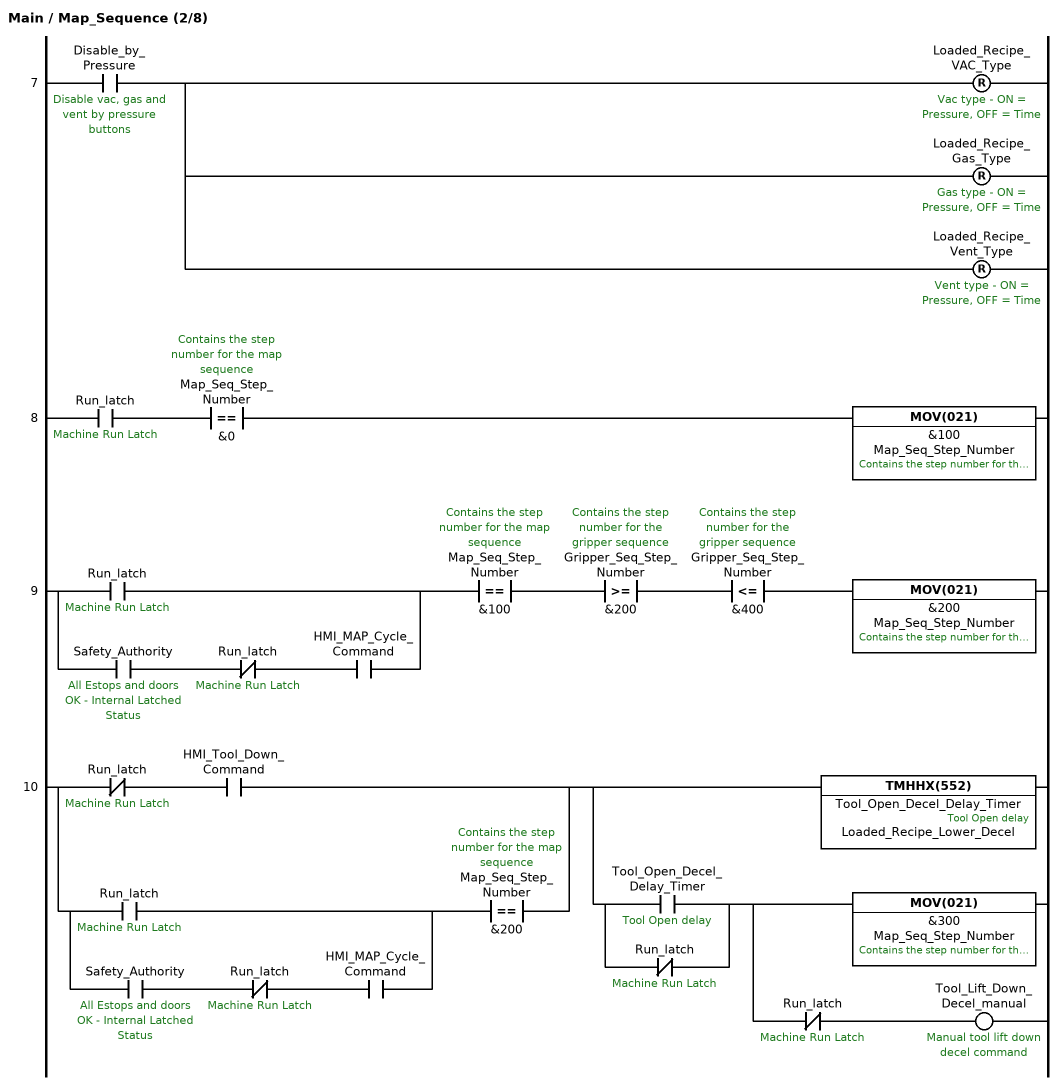
; rung 7
LD Disable_by_Pressure  ; Disable vac, gas and vent by pressure buttons
RSET Loaded_Recipe_VAC_Type  ; Vac type - ON = Pressure, OFF = Time
RSET Loaded_Recipe_Gas_Type  ; Gas type - ON = Pressure, OFF = Time
RSET Loaded_Recipe_Vent_Type  ; Vent type - ON = Pressure, OFF = Time
; rung 8
LD Run_latch  ; Machine Run Latch
AND=(300) Map_Seq_Step_Number &0  ; Contains the step number for the map sequence
MOV(021) &100 Map_Seq_Step_Number  ; Contains the step number for the map sequence
; rung 9
LD Run_latch  ; Machine Run Latch
LD Safety_Authority  ; All Estops and doors OK - Internal Latched Status
ANDNOT Run_latch  ; Machine Run Latch
AND HMI_MAP_Cycle_Command
ORLD
AND=(300) Map_Seq_Step_Number &100  ; Contains the step number for the map sequence
AND>=(325) Gripper_Seq_Step_Number &200  ; Contains the step number for the gripper sequence
AND<=(315) Gripper_Seq_Step_Number &400  ; Contains the step number for the gripper sequence
MOV(021) &200 Map_Seq_Step_Number  ; Contains the step number for the map sequence
; rung 10
LDNOT Run_latch  ; Machine Run Latch
AND HMI_Tool_Down_Command
LD Run_latch  ; Machine Run Latch
LD Safety_Authority  ; All Estops and doors OK - Internal Latched Status
ANDNOT Run_latch  ; Machine Run Latch
AND HMI_MAP_Cycle_Command
ORLD
AND=(300) Map_Seq_Step_Number &200  ; Contains the step number for the map sequence
ORLD
TMHHX(552) Tool_Open_Decel_Delay_Timer Loaded_Recipe_Lower_Decel  ; Tool Open delay
LD Tool_Open_Decel_Delay_Timer  ; Tool Open delay
ORNOT Run_latch  ; Machine Run Latch
ANDLD
MOV(021) &300 Map_Seq_Step_Number  ; Contains the step number for the map sequence
ANDNOT Run_latch  ; Machine Run Latch
OUT Tool_Lift_Down_Decel_manual  ; Manual tool lift down decel command

